FUNCTION_BLOCK FB_MY_BLINK
VAR_INPUT
	bEn : BOOL;
	udiTiOn_ms : UDINT := 100;
	udiTiOff_ms : UDINT := 100;
END_VAR
VAR_OUTPUT
	bQ : BOOL;
END_VAR
VAR
	state : WORD := 0;
	enTiOn : BOOL := FALSE;
	TiOn : TON;
	enTiOff : BOOL := FALSE;
	TiOff : TON;
END_VAR

CASE state OF
	0:
		IF bEn THEN
			state := 1;
			enTiOn := TRUE;
			bQ := TRUE;
		END_IF
	1:
		IF TiOn.Q THEN
			bQ := FALSE;
			enTiOn := FALSE;
			IF bEn THEN
				state := 2;
				enTiOff := TRUE;
			ELSE	
				state := 0;		
				enTiOff := FALSE;
			END_IF
		END_IF
	2:
		IF TiOff.Q THEN
			enTiOff := FALSE;
			IF bEn THEN
				state := 1;
				enTiOn := TRUE;
				bQ := TRUE;
			ELSE
				state := 0;
				enTiOn := FALSE;
				bQ := FALSE;
			END_IF
		END_IF
END_CASE
	
TiOn(IN := enTiOn, PT := UDINT_TO_TIME(udiTiOn_ms));

TiOff(IN := enTiOff, PT := UDINT_TO_TIME(udiTiOff_ms));

END_FUNCTION_BLOCK

(* stored: Version 1.1.0.1, ProductVersion 3.1.4024.3
   POU FB_MY_BLINK: Id {bfb42936-b033-4ca7-8b48-9f9bdb785ea8}, SpecialFunc None *)
